ABB RAPID module: input file 1

MODULE Module1
CONST robtarget Target_10:=[[869.327414578,176.772302874,635.169636394],[0.050595214,-0.000000043,0.998719242,-0.000000026],[0,-1,0,0],[9E+09,9E+09,9E+09,9E+09,9E+09,9E+09]];
CONST robtarget Target_20:=[[869.327418823,176.772296607,536.949239047],[0.050595245,-0.00000004,0.99871924,-0.000000026],[0,-1,0,0],[9E+09,9E+09,9E+09,9E+09,9E+09,9E+09]];
CONST robtarget Target_30:=[[869.327421447,176.772292534,624.0844316],[0.050595282,-0.000000037,0.998719239,-0.000000019],[0,-1,0,0],[9E+09,9E+09,9E+09,9E+09,9E+09,9E+09]];
CONST robtarget Target_40:=[[1343.783932622,176.772294127,624.084416899],[0.050595304,-0.000000028,0.998719237,-0.000000006],[0,-1,0,0],[9E+09,9E+09,9E+09,9E+09,9E+09,9E+09]];
CONST robtarget Target_50:=[[1343.783948564,176.772293806,510.50254946],[0.05059535,-0.000000026,0.998719235,0],[0,-1,0,0],[9E+09,9E+09,9E+09,9E+09,9E+09,9E+09]];
CONST robtarget Target_60:=[[1343.783944301,226.809597437,599.364401759],[0.050595404,-0.000000056,0.998719232,-0.000000053],[0,-1,0,0],[9E+09,9E+09,9E+09,9E+09,9E+09,9E+09]];
CONST robtarget Target_70:=[[1343.783935402,-246.064596292,594.1286137],[0.050595463,-0.000000068,0.998719229,-0.000000066],[-1,0,-1,0],[9E+09,9E+09,9E+09,9E+09,9E+09,9E+09]];
CONST robtarget Target_80:=[[1343.783944853,-246.064591904,505.19981437],[0.050595494,-0.000000065,0.998719228,-0.000000061],[-1,0,-1,0],[9E+09,9E+09,9E+09,9E+09,9E+09,9E+09]];
CONST robtarget Target_90:=[[1343.783949759,-261.778861424,591.432584085],[0.050595557,-0.000000098,0.998719225,-0.000000096],[-1,0,-1,0],[9E+09,9E+09,9E+09,9E+09,9E+09,9E+09]];
CONST robtarget Target_100:=[[918.872459934,-261.778889593,605.401239235],[0.050595633,-0.000000096,0.998719221,-0.000000097],[-1,0,-1,0],[9E+09,9E+09,9E+09,9E+09,9E+09,9E+09]];
CONST robtarget Target_110:=[[918.872450654,-261.778882858,516.455294008],[0.05059565,-0.000000098,0.99871922,-0.000000102],[-1,0,-1,0],[9E+09,9E+09,9E+09,9E+09,9E+09,9E+09]];
CONST robtarget Target_120:=[[918.872462038,-261.778863725,614.457432065],[0.050595676,-0.000000089,0.998719219,-0.000000069],[-1,0,-1,0],[9E+09,9E+09,9E+09,9E+09,9E+09,9E+09]];
CONST robtarget Target_130:=[[918.872477191,192.078304988,614.457463501],[0.050595717,-0.000000097,0.998719217,-0.000000075],[0,-1,0,0],[9E+09,9E+09,9E+09,9E+09,9E+09,9E+09]];
CONST robtarget Target_140:=[[918.872384855,14.98185962,963.600866633],[0.050595816,-0.000000108,0.998719211,-0.000000083],[0,-1,0,0],[9E+09,9E+09,9E+09,9E+09,9E+09,9E+09]];
CONST robtarget Target_140_2:=[[918.872384855,14.98185962,963.600866633],[0.050595816,-0.000000108,0.998719211,-0.000000083],[0,-1,0,0],[9E+09,9E+09,9E+09,9E+09,9E+09,9E+09]];
CONST robtarget Target_130_2:=[[918.872477191,192.078304988,614.457463501],[0.050595717,-0.000000097,0.998719217,-0.000000075],[0,-1,0,0],[9E+09,9E+09,9E+09,9E+09,9E+09,9E+09]];
CONST robtarget Target_120_2:=[[918.872462038,-261.778863725,614.457432065],[0.050595676,-0.000000089,0.998719219,-0.000000069],[-1,0,-1,0],[9E+09,9E+09,9E+09,9E+09,9E+09,9E+09]];
CONST robtarget Target_110_2:=[[918.872450654,-261.778882858,516.455294008],[0.05059565,-0.000000098,0.99871922,-0.000000102],[-1,0,-1,0],[9E+09,9E+09,9E+09,9E+09,9E+09,9E+09]];
CONST robtarget Target_100_2:=[[918.872459934,-261.778889593,605.401239235],[0.050595633,-0.000000096,0.998719221,-0.000000097],[-1,0,-1,0],[9E+09,9E+09,9E+09,9E+09,9E+09,9E+09]];
CONST robtarget Target_90_2:=[[1343.783949759,-261.778861424,591.432584085],[0.050595557,-0.000000098,0.998719225,-0.000000096],[-1,0,-1,0],[9E+09,9E+09,9E+09,9E+09,9E+09,9E+09]];
CONST robtarget Target_80_2:=[[1343.783944853,-246.064591904,505.19981437],[0.050595494,-0.000000065,0.998719228,-0.000000061],[-1,0,-1,0],[9E+09,9E+09,9E+09,9E+09,9E+09,9E+09]];
CONST robtarget Target_70_2:=[[1343.783935402,-246.064596292,594.1286137],[0.050595463,-0.000000068,0.998719229,-0.000000066],[-1,0,-1,0],[9E+09,9E+09,9E+09,9E+09,9E+09,9E+09]];
CONST robtarget Target_60_2:=[[1343.783944301,226.809597437,599.364401759],[0.050595404,-0.000000056,0.998719232,-0.000000053],[0,-1,0,0],[9E+09,9E+09,9E+09,9E+09,9E+09,9E+09]];
CONST robtarget Target_50_2:=[[1343.783948564,176.772293806,510.50254946],[0.05059535,-0.000000026,0.998719235,0],[0,-1,0,0],[9E+09,9E+09,9E+09,9E+09,9E+09,9E+09]];
CONST robtarget Target_40_2:=[[1343.783932622,176.772294127,624.084416899],[0.050595304,-0.000000028,0.998719237,-0.000000006],[0,-1,0,0],[9E+09,9E+09,9E+09,9E+09,9E+09,9E+09]];
CONST robtarget Target_30_2:=[[869.327421447,176.772292534,624.0844316],[0.050595282,-0.000000037,0.998719239,-0.000000019],[0,-1,0,0],[9E+09,9E+09,9E+09,9E+09,9E+09,9E+09]];
CONST robtarget Target_20_2:=[[869.327418823,176.772296607,536.949239047],[0.050595245,-0.00000004,0.99871924,-0.000000026],[0,-1,0,0],[9E+09,9E+09,9E+09,9E+09,9E+09,9E+09]];
CONST robtarget Target_10_2:=[[869.327414578,176.772302874,635.169636394],[0.050595214,-0.000000043,0.998719242,-0.000000026],[0,-1,0,0],[9E+09,9E+09,9E+09,9E+09,9E+09,9E+09]];
CONST robtarget Target_10_3:=[[869.327414578,176.772302874,635.169636394],[0.050595214,-0.000000043,0.998719242,-0.000000026],[0,-1,0,0],[9E+09,9E+09,9E+09,9E+09,9E+09,9E+09]];
CONST robtarget Target_20_3:=[[869.327418823,176.772296607,536.949239047],[0.050595245,-0.00000004,0.99871924,-0.000000026],[0,-1,0,0],[9E+09,9E+09,9E+09,9E+09,9E+09,9E+09]];
CONST robtarget Target_10_3_2:=[[869.327414578,176.772302874,635.169636394],[0.050595214,-0.000000043,0.998719242,-0.000000026],[0,-1,0,0],[9E+09,9E+09,9E+09,9E+09,9E+09,9E+09]];
CONST robtarget Target_20_3_2:=[[869.327418823,176.772296607,536.949239047],[0.050595245,-0.00000004,0.99871924,-0.000000026],[0,-1,0,0],[9E+09,9E+09,9E+09,9E+09,9E+09,9E+09]];
PERS num count :=0;
PROC main()
IF count>= 3 THEN
change_paper;
count:=0;
ENDIF
IF di1 =1 THEN
sharpen_pencil;
ENDIF
ENDPROC
PROC change_paper()
VAR num answer;
TPReadFK answer, "Change the paper", "OK", stEmpty, stEmpty,stEmpty, stEmpty;
ENDPROC
PROC sharpen_pencil()
SetDO do10,1;
MoveL Target_10_3,v100,z1,AW_Gun\WObj:=wobj0;
MoveL Target_20_3,v100,z5,AW_Gun\WObj:=wobj0;
MoveL Target_10_3_2,v100,z1,AW_Gun\WObj:=wobj0;
MoveL Target_20_3_2,v100,z5,AW_Gun\WObj:=wobj0;
SetDO do10,0;
ENDPROC
ENDMODULE
